FUNCTION_BLOCK fbRecorderRunnerTests
VAR
    _recorder : stRecorder;
END_VAR

{attribute 'TcRpcEnable'}
METHOD ResetCounter : UINT
_recorder.counter := 0;
END_METHOD

{attribute 'TcRpcEnable'}
METHOD RunWithRecorder : INT
RunWithRecorder := _recorder.counter;
END_METHOD

END_FUNCTION_BLOCK

(* stored: Version 1.1.0.1, ProductVersion 3.1.4024.6
   POU fbRecorderRunnerTests: Id {00761f1f-400a-4359-962b-f4cbcfef3f3d}, SpecialFunc None
   Method ResetCounter: Id {b3eccfe1-8058-4668-b649-6bc81b3eb643}
   Method RunWithRecorder: Id {e06617b6-3fea-491c-879a-664266fc030e} *)
